{attribute 'linkalways'} 
{attribute 'no_explicit_call' := 'This FB is a CLASS and must be accessed using methods or properties'}
{attribute 'enable_dynamic_creation'}
FUNCTION_BLOCK Node_F_VN_InvertAffineTransformation EXTENDS VisionNode
VAR
    aTransformationMatrix : _TcVnMatrix2x3_LREAL;
    aInvertedTransformationMatrix : _TcVnMatrix2x3_LREAL;
    hrPrev : _HRESULT(S_OK);
	hresult : _HRESULT(S_OK);
END_VAR

METHOD PUBLIC  Clone : I_Node
VAR
	pNode : POINTER TO Node_F_VN_InvertAffineTransformation;
END_VAR
pNode := __NEW(Node_F_VN_InvertAffineTransformation);
Clone := pNode^;
END_METHOD

METHOD FB_init : BOOL
VAR_INPUT
	bInitRetains : BOOL; // if TRUE, the retain variables are initialized (warm start / cold start)
	bInCopyCode : BOOL;  // if TRUE, the instance afterwards gets moved into the copy code (online change)
END_VAR
AddInput('aTransformationMatrix', aTransformationMatrix);
AddInput('hrPrev', hrPrev);
AddOutput('aInvertedTransformationMatrix', aInvertedTransformationMatrix);
AddOutput('hresult',hresult);
END_METHOD

METHOD PROTECTED  OnExecute : HRESULT
hresult.Value := F_VN_InvertAffineTransformation(
	aTransformationMatrix := aTransformationMatrix.Value,
    aInvertedTransformationMatrix := aInvertedTransformationMatrix.Value,
	hrPrev := hrPrev.Value);
END_METHOD

METHOD PUBLIC PreExecutionCheck
VAR_INPUT
	Check : I_PreExecutionChecks;
END_VAR
END_METHOD

END_FUNCTION_BLOCK

(* stored: Version 1.1.0.1, ProductVersion 3.1.4024.13
   POU Node_F_VN_InvertAffineTransformation: Id {2b14e65e-0a41-0e63-1bfa-bab5bff8b74a}, SpecialFunc None
   Folder Constructor: Id {f8caecf8-2463-0479-035a-7457abadd8f2}
   Method Clone: Id {382b6ff6-169d-006d-284c-764740ca3f49}
   Method FB_init: Id {7fbc4e4a-eb99-0fda-019b-a7022a176fbd}
   Method OnExecute: Id {98569669-835d-0492-1655-5d0a0f66d3d0}
   Method PreExecutionCheck: Id {a44b628a-7b5d-0db5-2775-abdc5e8a1dec} *)
